TYPE E_CalibrationState : (
    CAL_STATE_IDLE := 0,
    CAL_STATE_PRECHECK := 10,
    CAL_STATE_ACTIVE := 20,
    CAL_STATE_VALIDATE := 30,
    CAL_STATE_COMPLETE := 40,
    CAL_STATE_FAILED := 100
); END_TYPE

(* stored: Version 1.1.0.1
   DUT E_CalibrationState: Id {E3000000-0000-4000-8000-000000000020} *)
